Staubli VAL3: remErrRemoteKey.pgx

program remErrRemoteKey(string& sReturn[] (dimensions=1))
begin
  // Error raised when a command times out
  //
  logMsg("call remRemoteKey")
  sReturn="ERROR 402"
  sReturn=sReturn+": Select Remote mode using the key box."
  putln(sReturn)
  logMsg(sReturn)
end
